// TIA Portal V17 export
// export: Created 2024-06-14T09:52:24.0418538Z, ExportSetting WithDefaults, DisplayName Totally Integrated Automation Portal, DisplayVersion V17, DisplayName TIA Portal Openness, DisplayVersion V17, DisplayName TIA Portal Version Control Interface, DisplayVersion V17, DisplayName Simotion SCOUT TIA, DisplayVersion 5.4.3.0, DisplayName SINAMICS Startdrive Advanced, DisplayVersion V17 SP1 Update 1, DisplayName SINAMICS Startdrive G110M, G120, G120C, G120D, G120P, G115D, DisplayVersion V17 SP1 Update 1, DisplayName SINAMICS Startdrive G130, G150, S120, S150, SINAMICS MV, S210, DisplayVersion V17 SP1 Update 1, DisplayName STEP 7 Professional, DisplayVersion V17, DisplayName STEP 7 Safety, DisplayVersion V17, DisplayName WinCC Professional, DisplayVersion V17
FUNCTION_BLOCK "TCP_STN4_STN2_FB"   // FB120, LAD
{ S7_Optimized_Access := 'TRUE' }
VERSION : 0.1
// stored: AutoNumber false, IsIECCheckEnabled false, IsRetainMemResEnabled false, MemoryReserve 100, SetENOAutomatically false, UDAEnableTagReadback false
   VAR_OUTPUT
      Modbus_Busy : Bool;
   END_VAR
   VAR_IN_OUT
      Mod_TCP_Setup : "Mod_TCP_Data";
      LPG_Fill_Data : "LPG_FILL_DATA";
   END_VAR
   VAR
      PStep_No : Struct
         MASTER_STEP_NO : "Master_Step_No";
      END_STRUCT;
      Write_Bit_Address : Int;
      TRIG : Array[1..100] of Bool;
      Mod_Master1_Req : Array[1..10] of Bool;
      Mod_Master2_REQ : Array[1..10] of Bool;
      Mod_Master3_REQ : Array[1..10] of Bool;
      Mod_Master4_REQ : Array[1..10] of Bool;
      Mod_Master5_REQ : Array[1..10] of Bool;
      Mod_Master6_REQ : Array[1..10] of Bool;
      Mas_Trig_Extn { S7_SetPoint := 'True'} : TOF_TIME;
      Tare_delay { S7_SetPoint := 'True'} : TON_TIME;
   END_VAR
   VAR_TEMP
      Modbus_request : Bool;
   END_VAR
   VAR_TEMP   // added for the SCL form of the ladder/FBD networks
      _w1 : Bool;
      _w2 : Bool;
      _w3 : Bool;
      _w4 : Bool;
      _w5 : Bool;
      _w6 : Bool;
   END_VAR
BEGIN

REGION Network 1: FILLING LINE-1 STATION-2
END_REGION

REGION Network 2: Write Master-1 Holding Register Request(Tare Weight Entry)
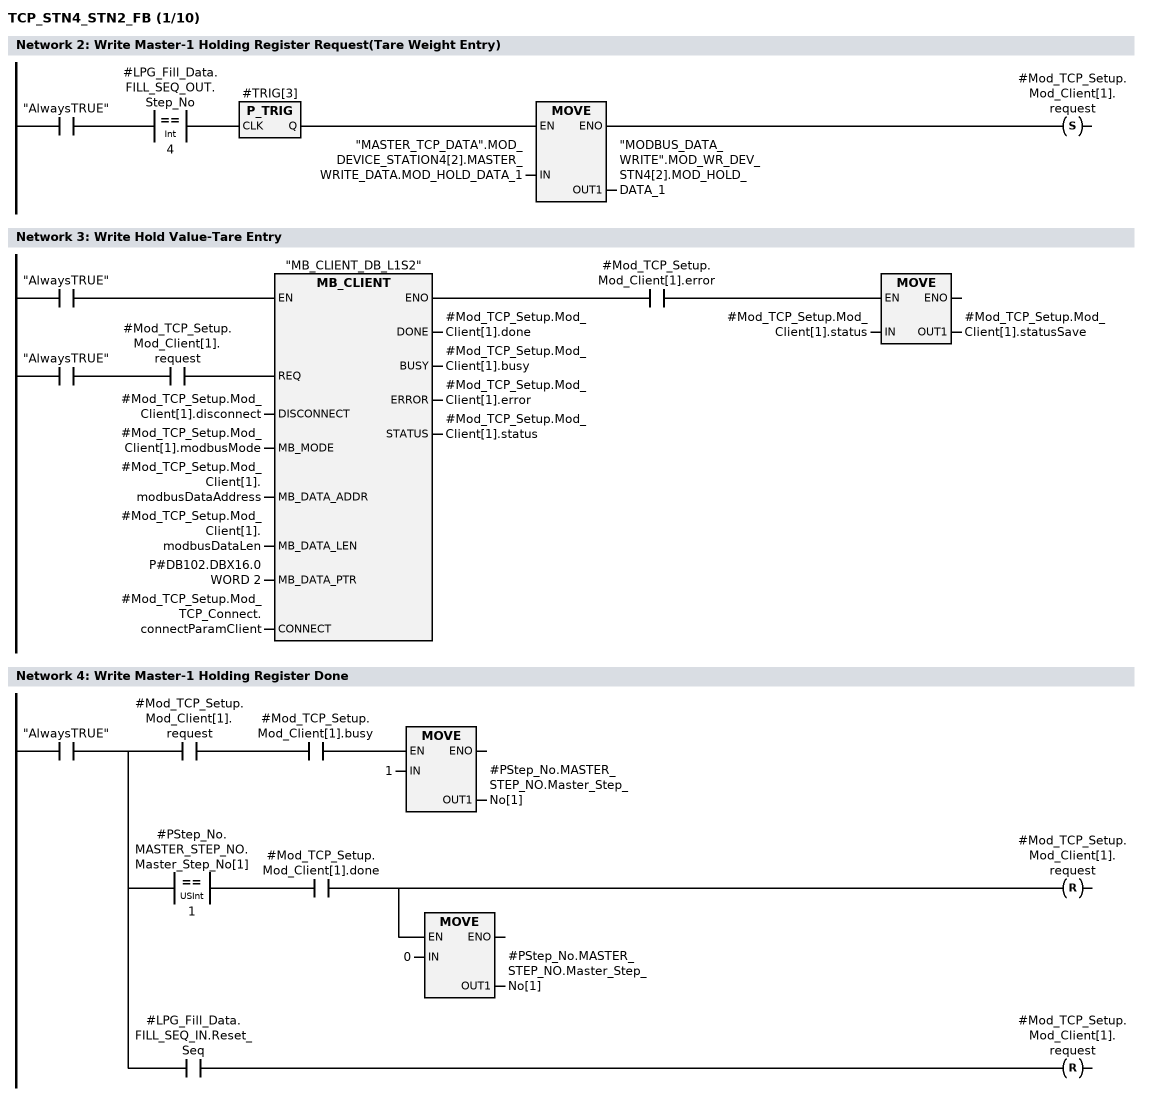
   RUNG wire#powerrail
      Contact( "AlwaysTRUE" )
      { S7_Templates := "SrcType := Int" } EQ_Contact(in1 := #LPG_Fill_Data.FILL_SEQ_OUT.Step_No, in2 := 4)
      P_Trig( #TRIG[3] )
      Move(in := "MASTER_TCP_DATA".MOD_DEVICE_STATION4[2].MASTER_WRITE_DATA.MOD_HOLD_DATA_1, out1 => "MODBUS_DATA_WRITE".MOD_WR_DEV_STN4[2].MOD_HOLD_DATA_1)
      S_Coil( #Mod_TCP_Setup.Mod_Client[1].request )
   END_RUNG
   // the same network as SCL:
   #_w1 := "AlwaysTRUE" AND (#LPG_Fill_Data.FILL_SEQ_OUT.Step_No = 4);
   #_w2 := #_w1 AND NOT #TRIG[3];   // rising edge
   #TRIG[3] := #_w1;
   IF #_w2 THEN
       "MODBUS_DATA_WRITE".MOD_WR_DEV_STN4[2].MOD_HOLD_DATA_1 := "MASTER_TCP_DATA".MOD_DEVICE_STATION4[2].MASTER_WRITE_DATA.MOD_HOLD_DATA_1;
       #Mod_TCP_Setup.Mod_Client[1].request := TRUE;
   END_IF;
END_REGION

REGION Network 3: Write Hold Value-Tare Entry
   RUNG wire#powerrail
      Contact( "AlwaysTRUE" )
      "MB_CLIENT_DB_L1S2".MB_CLIENT(REQ := wire#w1, DISCONNECT := #Mod_TCP_Setup.Mod_Client[1].disconnect, MB_MODE := #Mod_TCP_Setup.Mod_Client[1].modbusMode, MB_DATA_ADDR := #Mod_TCP_Setup.Mod_Client[1].modbusDataAddress, MB_DATA_LEN := #Mod_TCP_Setup.Mod_Client[1].modbusDataLen, MB_DATA_PTR := P#DB102.DBX16.0 WORD 2, CONNECT := #Mod_TCP_Setup.Mod_TCP_Connect.connectParamClient, DONE => #Mod_TCP_Setup.Mod_Client[1].done, BUSY => #Mod_TCP_Setup.Mod_Client[1].busy, ERROR => #Mod_TCP_Setup.Mod_Client[1].error, STATUS => #Mod_TCP_Setup.Mod_Client[1].status)
      Contact( #Mod_TCP_Setup.Mod_Client[1].error )
      Move(in := #Mod_TCP_Setup.Mod_Client[1].status, out1 => #Mod_TCP_Setup.Mod_Client[1].statusSave)
   END_RUNG
   RUNG wire#powerrail
      Contact( "AlwaysTRUE" )
      Contact( #Mod_TCP_Setup.Mod_Client[1].request )
   END_RUNG wire#w1
   // the same network as SCL:
   "MB_CLIENT_DB_L1S2"(EN := "AlwaysTRUE",   // MB_CLIENT
                       REQ := "AlwaysTRUE" AND #Mod_TCP_Setup.Mod_Client[1].request,
                       DISCONNECT := #Mod_TCP_Setup.Mod_Client[1].disconnect,
                       MB_MODE := #Mod_TCP_Setup.Mod_Client[1].modbusMode,
                       MB_DATA_ADDR := #Mod_TCP_Setup.Mod_Client[1].modbusDataAddress,
                       MB_DATA_LEN := #Mod_TCP_Setup.Mod_Client[1].modbusDataLen,
                       MB_DATA_PTR := P#DB102.DBX16.0 WORD 2,
                       CONNECT := #Mod_TCP_Setup.Mod_TCP_Connect.connectParamClient,
                       DONE => #Mod_TCP_Setup.Mod_Client[1].done,
                       BUSY => #Mod_TCP_Setup.Mod_Client[1].busy,
                       ERROR => #Mod_TCP_Setup.Mod_Client[1].error,
                       STATUS => #Mod_TCP_Setup.Mod_Client[1].status,
                       ENO => #_w1);
   IF #_w1 AND #Mod_TCP_Setup.Mod_Client[1].error THEN
       #Mod_TCP_Setup.Mod_Client[1].statusSave := #Mod_TCP_Setup.Mod_Client[1].status;
   END_IF;
END_REGION

REGION Network 4: Write Master-1 Holding Register Done
   RUNG wire#powerrail
      Contact( "AlwaysTRUE" )
      wire#w1
      Contact( #Mod_TCP_Setup.Mod_Client[1].request )
      Contact( #Mod_TCP_Setup.Mod_Client[1].busy )
      Move(in := 1, out1 => #PStep_No.MASTER_STEP_NO.Master_Step_No[1])
   END_RUNG
   RUNG wire#w1
      { S7_Templates := "SrcType := USInt" } EQ_Contact(in1 := #PStep_No.MASTER_STEP_NO.Master_Step_No[1], in2 := 1)
      Contact( #Mod_TCP_Setup.Mod_Client[1].done )
      wire#w2
      R_Coil( #Mod_TCP_Setup.Mod_Client[1].request )
   END_RUNG
   RUNG wire#w2
      Move(in := 0, out1 => #PStep_No.MASTER_STEP_NO.Master_Step_No[1])
   END_RUNG
   RUNG wire#w1
      Contact( #LPG_Fill_Data.FILL_SEQ_IN.Reset_Seq )
      R_Coil( #Mod_TCP_Setup.Mod_Client[1].request )
   END_RUNG
   // the same network as SCL:
   IF "AlwaysTRUE" AND #Mod_TCP_Setup.Mod_Client[1].request AND #Mod_TCP_Setup.Mod_Client[1].busy THEN
       #PStep_No.MASTER_STEP_NO.Master_Step_No[1] := 1;
   END_IF;
   #_w1 := "AlwaysTRUE" AND (#PStep_No.MASTER_STEP_NO.Master_Step_No[1] = 1) AND #Mod_TCP_Setup.Mod_Client[1].done;
   IF #_w1 THEN
       #Mod_TCP_Setup.Mod_Client[1].request := FALSE;
       #PStep_No.MASTER_STEP_NO.Master_Step_No[1] := 0;
   END_IF;
   IF "AlwaysTRUE" AND #LPG_Fill_Data.FILL_SEQ_IN.Reset_Seq THEN
       #Mod_TCP_Setup.Mod_Client[1].request := FALSE;
   END_IF;
END_REGION

REGION Network 5: Modbus Master2 Read Request(Filled Data)
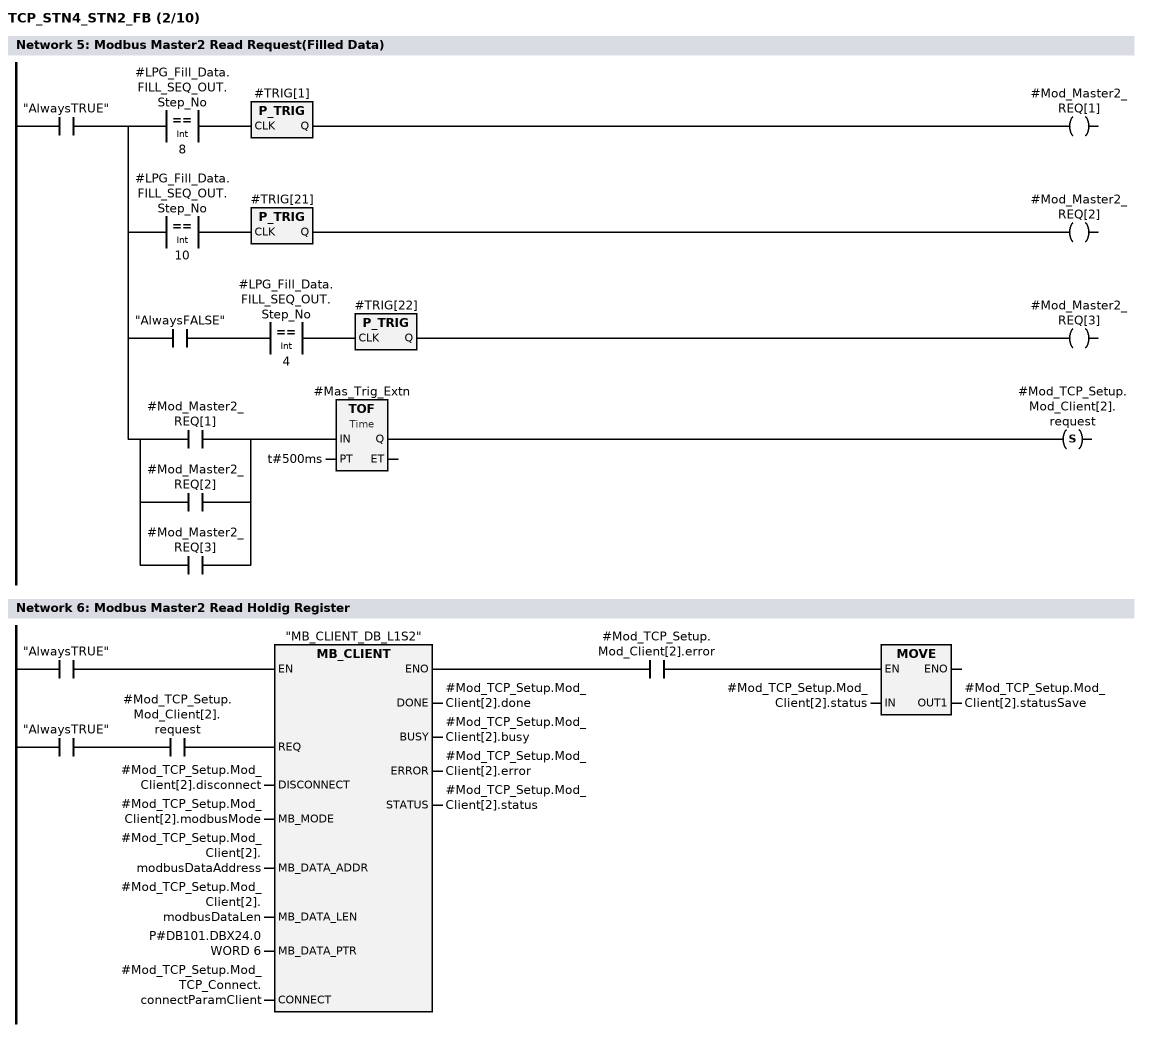
   RUNG wire#powerrail
      Contact( "AlwaysTRUE" )
      wire#w1
      { S7_Templates := "SrcType := Int" } EQ_Contact(in1 := #LPG_Fill_Data.FILL_SEQ_OUT.Step_No, in2 := 8)
      P_Trig( #TRIG[1] )
      Coil( #Mod_Master2_REQ[1] )
   END_RUNG
   RUNG wire#w1
      { S7_Templates := "SrcType := Int" } EQ_Contact(in1 := #LPG_Fill_Data.FILL_SEQ_OUT.Step_No, in2 := 10)
      P_Trig( #TRIG[21] )
      Coil( #Mod_Master2_REQ[2] )
   END_RUNG
   RUNG wire#w1
      Contact( "AlwaysFALSE" )
      { S7_Templates := "SrcType := Int" } EQ_Contact(in1 := #LPG_Fill_Data.FILL_SEQ_OUT.Step_No, in2 := 4)
      P_Trig( #TRIG[22] )
      Coil( #Mod_Master2_REQ[3] )
   END_RUNG
   RUNG wire#w1
      Contact( #Mod_Master2_REQ[1] )
      wire#w2
      { S7_Templates := "time_type := Time" } #Mas_Trig_Extn.TOF(pt := t#500ms, et =>)
      S_Coil( #Mod_TCP_Setup.Mod_Client[2].request )
   END_RUNG
   RUNG wire#w1
      Contact( #Mod_Master2_REQ[2] )
   END_RUNG wire#w2
   RUNG wire#w1
      Contact( #Mod_Master2_REQ[3] )
   END_RUNG wire#w2
   // the same network as SCL:
   #_w1 := "AlwaysTRUE" AND (#LPG_Fill_Data.FILL_SEQ_OUT.Step_No = 8);
   #_w2 := #_w1 AND NOT #TRIG[1];   // rising edge
   #TRIG[1] := #_w1;
   #Mod_Master2_REQ[1] := #_w2;
   #_w3 := "AlwaysTRUE" AND (#LPG_Fill_Data.FILL_SEQ_OUT.Step_No = 10);
   #_w4 := #_w3 AND NOT #TRIG[21];   // rising edge
   #TRIG[21] := #_w3;
   #Mod_Master2_REQ[2] := #_w4;
   #_w5 := "AlwaysTRUE" AND "AlwaysFALSE" AND (#LPG_Fill_Data.FILL_SEQ_OUT.Step_No = 4);
   #_w6 := #_w5 AND NOT #TRIG[22];   // rising edge
   #TRIG[22] := #_w5;
   #Mod_Master2_REQ[3] := #_w6;
   #Mas_Trig_Extn(IN := "AlwaysTRUE" AND (#Mod_Master2_REQ[1] OR #Mod_Master2_REQ[2] OR #Mod_Master2_REQ[3]),   // TOF
                  PT := t#500ms);
   IF #Mas_Trig_Extn.Q THEN #Mod_TCP_Setup.Mod_Client[2].request := TRUE; END_IF;
END_REGION

REGION Network 6: Modbus Master2 Read Holdig Register
   RUNG wire#powerrail
      Contact( "AlwaysTRUE" )
      "MB_CLIENT_DB_L1S2".MB_CLIENT(REQ := wire#w1, DISCONNECT := #Mod_TCP_Setup.Mod_Client[2].disconnect, MB_MODE := #Mod_TCP_Setup.Mod_Client[2].modbusMode, MB_DATA_ADDR := #Mod_TCP_Setup.Mod_Client[2].modbusDataAddress, MB_DATA_LEN := #Mod_TCP_Setup.Mod_Client[2].modbusDataLen, MB_DATA_PTR := P#DB101.DBX24.0 WORD 6, CONNECT := #Mod_TCP_Setup.Mod_TCP_Connect.connectParamClient, DONE => #Mod_TCP_Setup.Mod_Client[2].done, BUSY => #Mod_TCP_Setup.Mod_Client[2].busy, ERROR => #Mod_TCP_Setup.Mod_Client[2].error, STATUS => #Mod_TCP_Setup.Mod_Client[2].status)
      Contact( #Mod_TCP_Setup.Mod_Client[2].error )
      Move(in := #Mod_TCP_Setup.Mod_Client[2].status, out1 => #Mod_TCP_Setup.Mod_Client[2].statusSave)
   END_RUNG
   RUNG wire#powerrail
      Contact( "AlwaysTRUE" )
      Contact( #Mod_TCP_Setup.Mod_Client[2].request )
   END_RUNG wire#w1
   // the same network as SCL:
   "MB_CLIENT_DB_L1S2"(EN := "AlwaysTRUE",   // MB_CLIENT
                       REQ := "AlwaysTRUE" AND #Mod_TCP_Setup.Mod_Client[2].request,
                       DISCONNECT := #Mod_TCP_Setup.Mod_Client[2].disconnect,
                       MB_MODE := #Mod_TCP_Setup.Mod_Client[2].modbusMode,
                       MB_DATA_ADDR := #Mod_TCP_Setup.Mod_Client[2].modbusDataAddress,
                       MB_DATA_LEN := #Mod_TCP_Setup.Mod_Client[2].modbusDataLen,
                       MB_DATA_PTR := P#DB101.DBX24.0 WORD 6,
                       CONNECT := #Mod_TCP_Setup.Mod_TCP_Connect.connectParamClient,
                       DONE => #Mod_TCP_Setup.Mod_Client[2].done,
                       BUSY => #Mod_TCP_Setup.Mod_Client[2].busy,
                       ERROR => #Mod_TCP_Setup.Mod_Client[2].error,
                       STATUS => #Mod_TCP_Setup.Mod_Client[2].status,
                       ENO => #_w1);
   IF #_w1 AND #Mod_TCP_Setup.Mod_Client[2].error THEN
       #Mod_TCP_Setup.Mod_Client[2].statusSave := #Mod_TCP_Setup.Mod_Client[2].status;
   END_IF;
END_REGION

REGION Network 7: Read Master-2 Holding Register Value
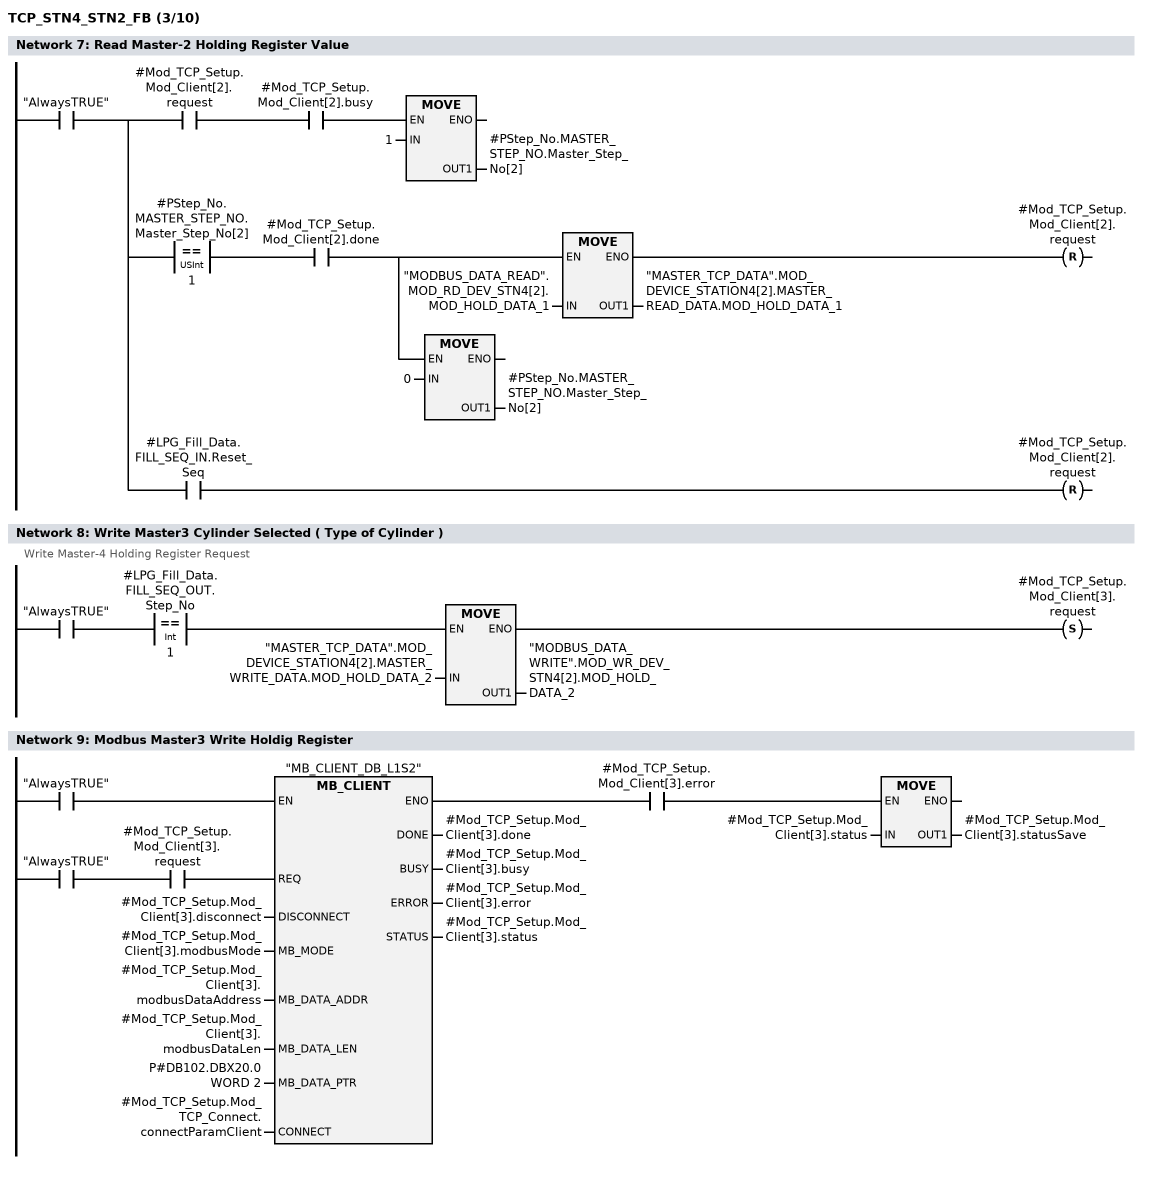
   RUNG wire#powerrail
      Contact( "AlwaysTRUE" )
      wire#w1
      Contact( #Mod_TCP_Setup.Mod_Client[2].request )
      Contact( #Mod_TCP_Setup.Mod_Client[2].busy )
      Move(in := 1, out1 => #PStep_No.MASTER_STEP_NO.Master_Step_No[2])
   END_RUNG
   RUNG wire#w1
      { S7_Templates := "SrcType := USInt" } EQ_Contact(in1 := #PStep_No.MASTER_STEP_NO.Master_Step_No[2], in2 := 1)
      Contact( #Mod_TCP_Setup.Mod_Client[2].done )
      wire#w2
      Move(in := "MODBUS_DATA_READ".MOD_RD_DEV_STN4[2].MOD_HOLD_DATA_1, out1 => "MASTER_TCP_DATA".MOD_DEVICE_STATION4[2].MASTER_READ_DATA.MOD_HOLD_DATA_1)
      R_Coil( #Mod_TCP_Setup.Mod_Client[2].request )
   END_RUNG
   RUNG wire#w2
      Move(in := 0, out1 => #PStep_No.MASTER_STEP_NO.Master_Step_No[2])
   END_RUNG
   RUNG wire#w1
      Contact( #LPG_Fill_Data.FILL_SEQ_IN.Reset_Seq )
      R_Coil( #Mod_TCP_Setup.Mod_Client[2].request )
   END_RUNG
   // the same network as SCL:
   IF "AlwaysTRUE" AND #Mod_TCP_Setup.Mod_Client[2].request AND #Mod_TCP_Setup.Mod_Client[2].busy THEN
       #PStep_No.MASTER_STEP_NO.Master_Step_No[2] := 1;
   END_IF;
   IF "AlwaysTRUE" AND (#PStep_No.MASTER_STEP_NO.Master_Step_No[2] = 1) AND #Mod_TCP_Setup.Mod_Client[2].done THEN
       "MASTER_TCP_DATA".MOD_DEVICE_STATION4[2].MASTER_READ_DATA.MOD_HOLD_DATA_1 := "MODBUS_DATA_READ".MOD_RD_DEV_STN4[2].MOD_HOLD_DATA_1;
   END_IF;
   #_w1 := "AlwaysTRUE" AND (#PStep_No.MASTER_STEP_NO.Master_Step_No[2] = 1) AND #Mod_TCP_Setup.Mod_Client[2].done;
   IF #_w1 THEN
       #Mod_TCP_Setup.Mod_Client[2].request := FALSE;
       #PStep_No.MASTER_STEP_NO.Master_Step_No[2] := 0;
   END_IF;
   IF "AlwaysTRUE" AND #LPG_Fill_Data.FILL_SEQ_IN.Reset_Seq THEN
       #Mod_TCP_Setup.Mod_Client[2].request := FALSE;
   END_IF;
END_REGION

REGION Network 8: Write Master3 Cylinder Selected ( Type of Cylinder )
   // Write Master-4 Holding Register Request
   RUNG wire#powerrail
      Contact( "AlwaysTRUE" )
      { S7_Templates := "SrcType := Int" } EQ_Contact(in1 := #LPG_Fill_Data.FILL_SEQ_OUT.Step_No, in2 := 1)
      Move(in := "MASTER_TCP_DATA".MOD_DEVICE_STATION4[2].MASTER_WRITE_DATA.MOD_HOLD_DATA_2, out1 => "MODBUS_DATA_WRITE".MOD_WR_DEV_STN4[2].MOD_HOLD_DATA_2)
      S_Coil( #Mod_TCP_Setup.Mod_Client[3].request )
   END_RUNG
   // the same network as SCL:
   IF "AlwaysTRUE" AND (#LPG_Fill_Data.FILL_SEQ_OUT.Step_No = 1) THEN
       "MODBUS_DATA_WRITE".MOD_WR_DEV_STN4[2].MOD_HOLD_DATA_2 := "MASTER_TCP_DATA".MOD_DEVICE_STATION4[2].MASTER_WRITE_DATA.MOD_HOLD_DATA_2;
       #Mod_TCP_Setup.Mod_Client[3].request := TRUE;
   END_IF;
END_REGION

REGION Network 9: Modbus Master3 Write Holdig Register
   RUNG wire#powerrail
      Contact( "AlwaysTRUE" )
      "MB_CLIENT_DB_L1S2".MB_CLIENT(REQ := wire#w1, DISCONNECT := #Mod_TCP_Setup.Mod_Client[3].disconnect, MB_MODE := #Mod_TCP_Setup.Mod_Client[3].modbusMode, MB_DATA_ADDR := #Mod_TCP_Setup.Mod_Client[3].modbusDataAddress, MB_DATA_LEN := #Mod_TCP_Setup.Mod_Client[3].modbusDataLen, MB_DATA_PTR := P#DB102.DBX20.0 WORD 2, CONNECT := #Mod_TCP_Setup.Mod_TCP_Connect.connectParamClient, DONE => #Mod_TCP_Setup.Mod_Client[3].done, BUSY => #Mod_TCP_Setup.Mod_Client[3].busy, ERROR => #Mod_TCP_Setup.Mod_Client[3].error, STATUS => #Mod_TCP_Setup.Mod_Client[3].status)
      Contact( #Mod_TCP_Setup.Mod_Client[3].error )
      Move(in := #Mod_TCP_Setup.Mod_Client[3].status, out1 => #Mod_TCP_Setup.Mod_Client[3].statusSave)
   END_RUNG
   RUNG wire#powerrail
      Contact( "AlwaysTRUE" )
      Contact( #Mod_TCP_Setup.Mod_Client[3].request )
   END_RUNG wire#w1
   // the same network as SCL:
   "MB_CLIENT_DB_L1S2"(EN := "AlwaysTRUE",   // MB_CLIENT
                       REQ := "AlwaysTRUE" AND #Mod_TCP_Setup.Mod_Client[3].request,
                       DISCONNECT := #Mod_TCP_Setup.Mod_Client[3].disconnect,
                       MB_MODE := #Mod_TCP_Setup.Mod_Client[3].modbusMode,
                       MB_DATA_ADDR := #Mod_TCP_Setup.Mod_Client[3].modbusDataAddress,
                       MB_DATA_LEN := #Mod_TCP_Setup.Mod_Client[3].modbusDataLen,
                       MB_DATA_PTR := P#DB102.DBX20.0 WORD 2,
                       CONNECT := #Mod_TCP_Setup.Mod_TCP_Connect.connectParamClient,
                       DONE => #Mod_TCP_Setup.Mod_Client[3].done,
                       BUSY => #Mod_TCP_Setup.Mod_Client[3].busy,
                       ERROR => #Mod_TCP_Setup.Mod_Client[3].error,
                       STATUS => #Mod_TCP_Setup.Mod_Client[3].status,
                       ENO => #_w1);
   IF #_w1 AND #Mod_TCP_Setup.Mod_Client[3].error THEN
       #Mod_TCP_Setup.Mod_Client[3].statusSave := #Mod_TCP_Setup.Mod_Client[3].status;
   END_IF;
END_REGION

REGION Network 10: Write Master-3 Holding Register Done
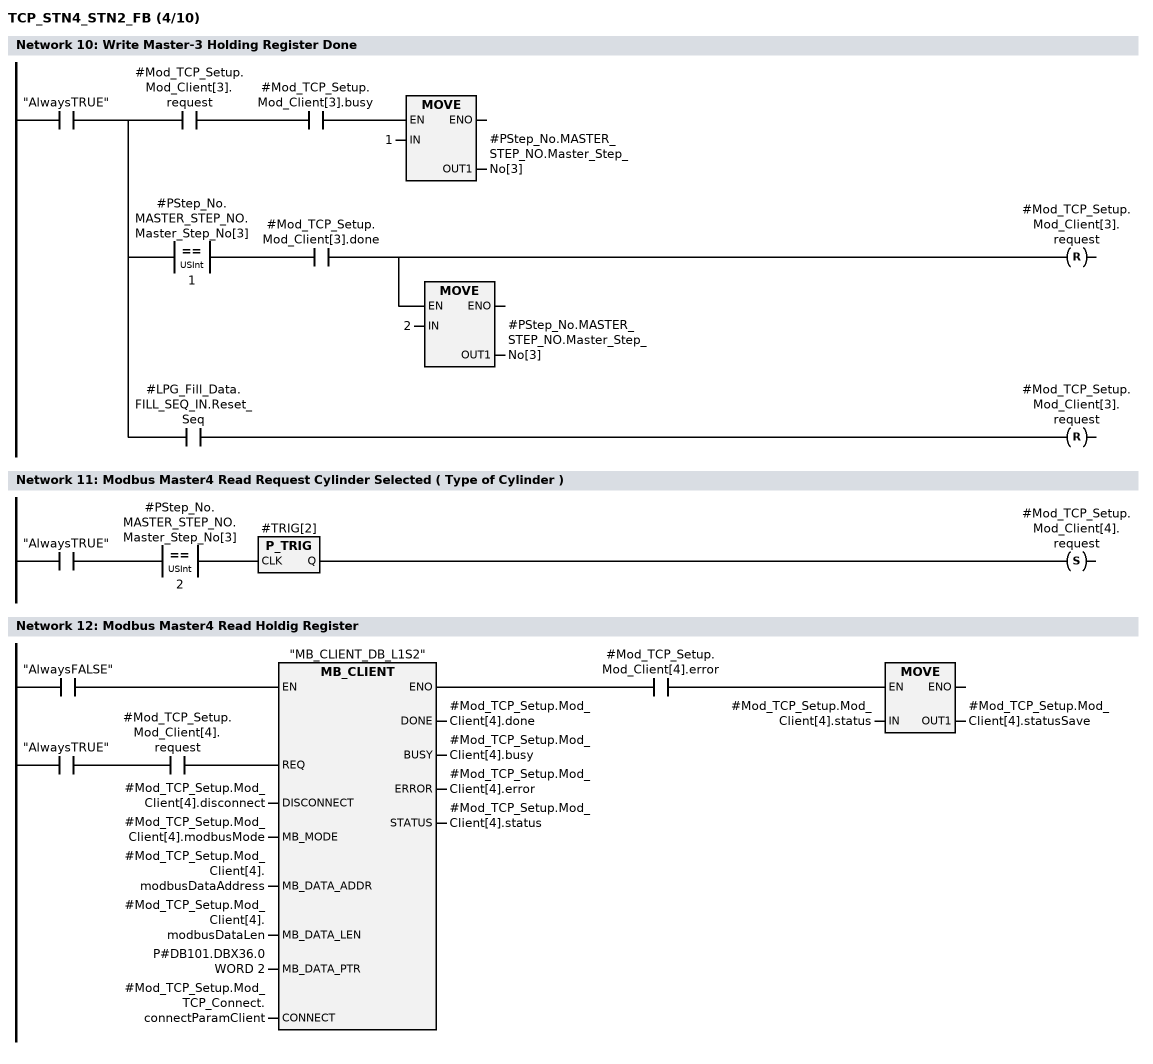
   RUNG wire#powerrail
      Contact( "AlwaysTRUE" )
      wire#w1
      Contact( #Mod_TCP_Setup.Mod_Client[3].request )
      Contact( #Mod_TCP_Setup.Mod_Client[3].busy )
      Move(in := 1, out1 => #PStep_No.MASTER_STEP_NO.Master_Step_No[3])
   END_RUNG
   RUNG wire#w1
      { S7_Templates := "SrcType := USInt" } EQ_Contact(in1 := #PStep_No.MASTER_STEP_NO.Master_Step_No[3], in2 := 1)
      Contact( #Mod_TCP_Setup.Mod_Client[3].done )
      wire#w2
      R_Coil( #Mod_TCP_Setup.Mod_Client[3].request )
   END_RUNG
   RUNG wire#w2
      Move(in := 2, out1 => #PStep_No.MASTER_STEP_NO.Master_Step_No[3])
   END_RUNG
   RUNG wire#w1
      Contact( #LPG_Fill_Data.FILL_SEQ_IN.Reset_Seq )
      R_Coil( #Mod_TCP_Setup.Mod_Client[3].request )
   END_RUNG
   // the same network as SCL:
   IF "AlwaysTRUE" AND #Mod_TCP_Setup.Mod_Client[3].request AND #Mod_TCP_Setup.Mod_Client[3].busy THEN
       #PStep_No.MASTER_STEP_NO.Master_Step_No[3] := 1;
   END_IF;
   #_w1 := "AlwaysTRUE" AND (#PStep_No.MASTER_STEP_NO.Master_Step_No[3] = 1) AND #Mod_TCP_Setup.Mod_Client[3].done;
   IF #_w1 THEN
       #Mod_TCP_Setup.Mod_Client[3].request := FALSE;
       #PStep_No.MASTER_STEP_NO.Master_Step_No[3] := 2;
   END_IF;
   IF "AlwaysTRUE" AND #LPG_Fill_Data.FILL_SEQ_IN.Reset_Seq THEN
       #Mod_TCP_Setup.Mod_Client[3].request := FALSE;
   END_IF;
END_REGION

REGION Network 11: Modbus Master4 Read Request Cylinder Selected ( Type of Cylinder )
   RUNG wire#powerrail
      Contact( "AlwaysTRUE" )
      { S7_Templates := "SrcType := USInt" } EQ_Contact(in1 := #PStep_No.MASTER_STEP_NO.Master_Step_No[3], in2 := 2)
      P_Trig( #TRIG[2] )
      S_Coil( #Mod_TCP_Setup.Mod_Client[4].request )
   END_RUNG
   // the same network as SCL:
   #_w1 := "AlwaysTRUE" AND (#PStep_No.MASTER_STEP_NO.Master_Step_No[3] = 2);
   #_w2 := #_w1 AND NOT #TRIG[2];   // rising edge
   #TRIG[2] := #_w1;
   IF #_w2 THEN #Mod_TCP_Setup.Mod_Client[4].request := TRUE; END_IF;
END_REGION

REGION Network 12: Modbus Master4 Read Holdig Register
   RUNG wire#powerrail
      Contact( "AlwaysFALSE" )
      "MB_CLIENT_DB_L1S2".MB_CLIENT(REQ := wire#w1, DISCONNECT := #Mod_TCP_Setup.Mod_Client[4].disconnect, MB_MODE := #Mod_TCP_Setup.Mod_Client[4].modbusMode, MB_DATA_ADDR := #Mod_TCP_Setup.Mod_Client[4].modbusDataAddress, MB_DATA_LEN := #Mod_TCP_Setup.Mod_Client[4].modbusDataLen, MB_DATA_PTR := P#DB101.DBX36.0 WORD 2, CONNECT := #Mod_TCP_Setup.Mod_TCP_Connect.connectParamClient, DONE => #Mod_TCP_Setup.Mod_Client[4].done, BUSY => #Mod_TCP_Setup.Mod_Client[4].busy, ERROR => #Mod_TCP_Setup.Mod_Client[4].error, STATUS => #Mod_TCP_Setup.Mod_Client[4].status)
      Contact( #Mod_TCP_Setup.Mod_Client[4].error )
      Move(in := #Mod_TCP_Setup.Mod_Client[4].status, out1 => #Mod_TCP_Setup.Mod_Client[4].statusSave)
   END_RUNG
   RUNG wire#powerrail
      Contact( "AlwaysTRUE" )
      Contact( #Mod_TCP_Setup.Mod_Client[4].request )
   END_RUNG wire#w1
   // the same network as SCL:
   "MB_CLIENT_DB_L1S2"(EN := "AlwaysFALSE",   // MB_CLIENT
                       REQ := "AlwaysTRUE" AND #Mod_TCP_Setup.Mod_Client[4].request,
                       DISCONNECT := #Mod_TCP_Setup.Mod_Client[4].disconnect,
                       MB_MODE := #Mod_TCP_Setup.Mod_Client[4].modbusMode,
                       MB_DATA_ADDR := #Mod_TCP_Setup.Mod_Client[4].modbusDataAddress,
                       MB_DATA_LEN := #Mod_TCP_Setup.Mod_Client[4].modbusDataLen,
                       MB_DATA_PTR := P#DB101.DBX36.0 WORD 2,
                       CONNECT := #Mod_TCP_Setup.Mod_TCP_Connect.connectParamClient,
                       DONE => #Mod_TCP_Setup.Mod_Client[4].done,
                       BUSY => #Mod_TCP_Setup.Mod_Client[4].busy,
                       ERROR => #Mod_TCP_Setup.Mod_Client[4].error,
                       STATUS => #Mod_TCP_Setup.Mod_Client[4].status,
                       ENO => #_w1);
   IF #_w1 AND #Mod_TCP_Setup.Mod_Client[4].error THEN
       #Mod_TCP_Setup.Mod_Client[4].statusSave := #Mod_TCP_Setup.Mod_Client[4].status;
   END_IF;
END_REGION

REGION Network 13: Read Master-4 Holding Register Value
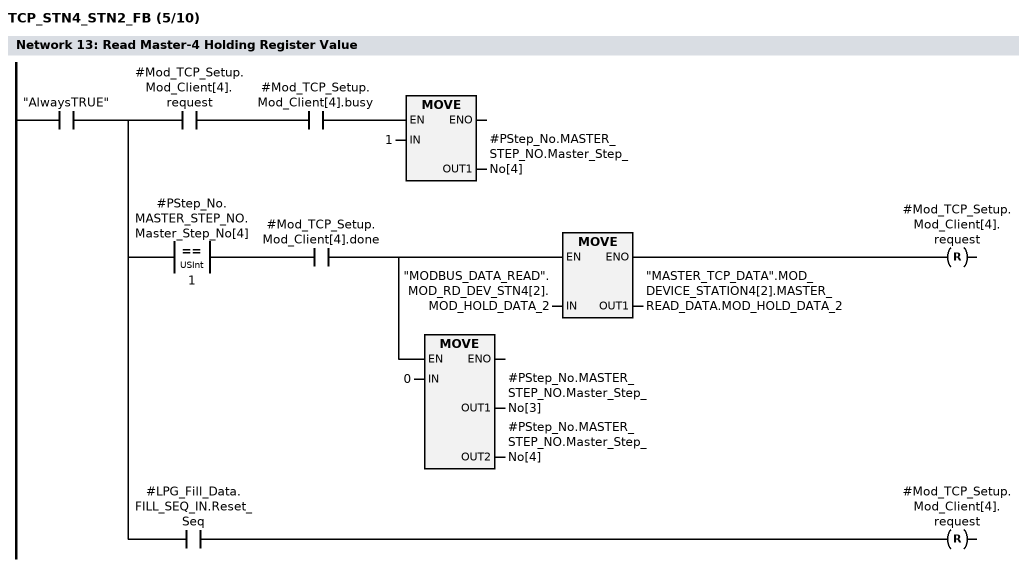
   RUNG wire#powerrail
      Contact( "AlwaysTRUE" )
      wire#w1
      Contact( #Mod_TCP_Setup.Mod_Client[4].request )
      Contact( #Mod_TCP_Setup.Mod_Client[4].busy )
      Move(in := 1, out1 => #PStep_No.MASTER_STEP_NO.Master_Step_No[4])
   END_RUNG
   RUNG wire#w1
      { S7_Templates := "SrcType := USInt" } EQ_Contact(in1 := #PStep_No.MASTER_STEP_NO.Master_Step_No[4], in2 := 1)
      Contact( #Mod_TCP_Setup.Mod_Client[4].done )
      wire#w2
      Move(in := "MODBUS_DATA_READ".MOD_RD_DEV_STN4[2].MOD_HOLD_DATA_2, out1 => "MASTER_TCP_DATA".MOD_DEVICE_STATION4[2].MASTER_READ_DATA.MOD_HOLD_DATA_2)
      R_Coil( #Mod_TCP_Setup.Mod_Client[4].request )
   END_RUNG
   RUNG wire#w2
      Move(in := 0, out1 => #PStep_No.MASTER_STEP_NO.Master_Step_No[3], out2 => #PStep_No.MASTER_STEP_NO.Master_Step_No[4])
   END_RUNG
   RUNG wire#w1
      Contact( #LPG_Fill_Data.FILL_SEQ_IN.Reset_Seq )
      R_Coil( #Mod_TCP_Setup.Mod_Client[4].request )
   END_RUNG
   // the same network as SCL:
   IF "AlwaysTRUE" AND #Mod_TCP_Setup.Mod_Client[4].request AND #Mod_TCP_Setup.Mod_Client[4].busy THEN
       #PStep_No.MASTER_STEP_NO.Master_Step_No[4] := 1;
   END_IF;
   IF "AlwaysTRUE" AND (#PStep_No.MASTER_STEP_NO.Master_Step_No[4] = 1) AND #Mod_TCP_Setup.Mod_Client[4].done THEN
       "MASTER_TCP_DATA".MOD_DEVICE_STATION4[2].MASTER_READ_DATA.MOD_HOLD_DATA_2 := "MODBUS_DATA_READ".MOD_RD_DEV_STN4[2].MOD_HOLD_DATA_2;
   END_IF;
   #_w1 := "AlwaysTRUE" AND (#PStep_No.MASTER_STEP_NO.Master_Step_No[4] = 1) AND #Mod_TCP_Setup.Mod_Client[4].done;
   IF #_w1 THEN
       #Mod_TCP_Setup.Mod_Client[4].request := FALSE;
       #PStep_No.MASTER_STEP_NO.Master_Step_No[3] := 0;
       #PStep_No.MASTER_STEP_NO.Master_Step_No[4] := 0;
   END_IF;
   IF "AlwaysTRUE" AND #LPG_Fill_Data.FILL_SEQ_IN.Reset_Seq THEN
       #Mod_TCP_Setup.Mod_Client[4].request := FALSE;
   END_IF;
END_REGION

REGION Network 14: Modbus Master5 Read Request(Coil Status)
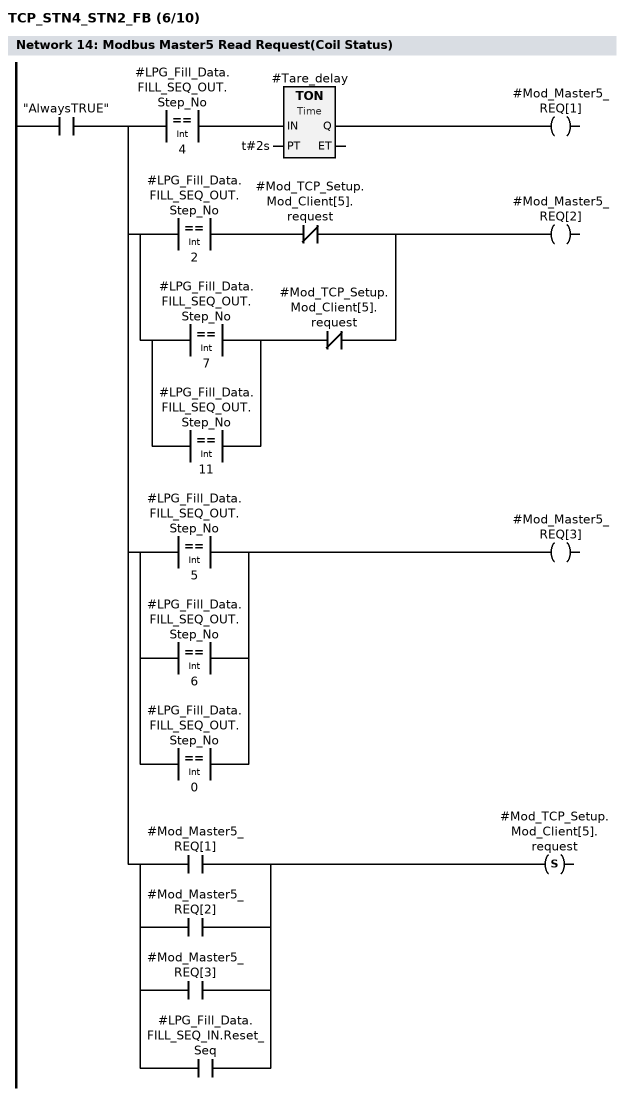
   RUNG wire#powerrail
      Contact( "AlwaysTRUE" )
      wire#w1
      { S7_Templates := "SrcType := Int" } EQ_Contact(in1 := #LPG_Fill_Data.FILL_SEQ_OUT.Step_No, in2 := 4)
      { S7_Templates := "time_type := Time" } #Tare_delay.TON(pt := t#2s, et =>)
      Coil( #Mod_Master5_REQ[1] )
   END_RUNG
   RUNG wire#w1
      { S7_Templates := "SrcType := Int" } EQ_Contact(in1 := #LPG_Fill_Data.FILL_SEQ_OUT.Step_No, in2 := 2)
      I_Contact( #Mod_TCP_Setup.Mod_Client[5].request )
      wire#w2
      Coil( #Mod_Master5_REQ[2] )
   END_RUNG
   RUNG wire#w1
      { S7_Templates := "SrcType := Int" } EQ_Contact(in1 := #LPG_Fill_Data.FILL_SEQ_OUT.Step_No, in2 := 7)
      wire#w3
      I_Contact( #Mod_TCP_Setup.Mod_Client[5].request )
   END_RUNG wire#w2
   RUNG wire#w1
      { S7_Templates := "SrcType := Int" } EQ_Contact(in1 := #LPG_Fill_Data.FILL_SEQ_OUT.Step_No, in2 := 11)
   END_RUNG wire#w3
   RUNG wire#w1
      { S7_Templates := "SrcType := Int" } EQ_Contact(in1 := #LPG_Fill_Data.FILL_SEQ_OUT.Step_No, in2 := 5)
      wire#w4
      Coil( #Mod_Master5_REQ[3] )
   END_RUNG
   RUNG wire#w1
      { S7_Templates := "SrcType := Int" } EQ_Contact(in1 := #LPG_Fill_Data.FILL_SEQ_OUT.Step_No, in2 := 6)
   END_RUNG wire#w4
   RUNG wire#w1
      { S7_Templates := "SrcType := Int" } EQ_Contact(in1 := #LPG_Fill_Data.FILL_SEQ_OUT.Step_No, in2 := 0)
   END_RUNG wire#w4
   RUNG wire#w1
      Contact( #Mod_Master5_REQ[1] )
      wire#w5
      S_Coil( #Mod_TCP_Setup.Mod_Client[5].request )
   END_RUNG
   RUNG wire#w1
      Contact( #Mod_Master5_REQ[2] )
   END_RUNG wire#w5
   RUNG wire#w1
      Contact( #Mod_Master5_REQ[3] )
   END_RUNG wire#w5
   RUNG wire#w1
      Contact( #LPG_Fill_Data.FILL_SEQ_IN.Reset_Seq )
   END_RUNG wire#w5
   // the same network as SCL:
   #Tare_delay(IN := "AlwaysTRUE" AND (#LPG_Fill_Data.FILL_SEQ_OUT.Step_No = 4), PT := t#2s);   // TON
   #Mod_Master5_REQ[1] := #Tare_delay.Q;
   #Mod_Master5_REQ[2] := "AlwaysTRUE" AND (((#LPG_Fill_Data.FILL_SEQ_OUT.Step_No = 2) AND NOT #Mod_TCP_Setup.Mod_Client[5].request) OR (((#LPG_Fill_Data.FILL_SEQ_OUT.Step_No = 7) OR (#LPG_Fill_Data.FILL_SEQ_OUT.Step_No = 11)) AND NOT #Mod_TCP_Setup.Mod_Client[5].request));
   #Mod_Master5_REQ[3] := "AlwaysTRUE" AND ((#LPG_Fill_Data.FILL_SEQ_OUT.Step_No = 5) OR (#LPG_Fill_Data.FILL_SEQ_OUT.Step_No = 6) OR (#LPG_Fill_Data.FILL_SEQ_OUT.Step_No = 0));
   IF "AlwaysTRUE" AND (#Mod_Master5_REQ[1] OR #Mod_Master5_REQ[2] OR #Mod_Master5_REQ[3] OR #LPG_Fill_Data.FILL_SEQ_IN.Reset_Seq) THEN
       #Mod_TCP_Setup.Mod_Client[5].request := TRUE;
   END_IF;
END_REGION

REGION Network 15: Modbus Master5 Read Coil Status
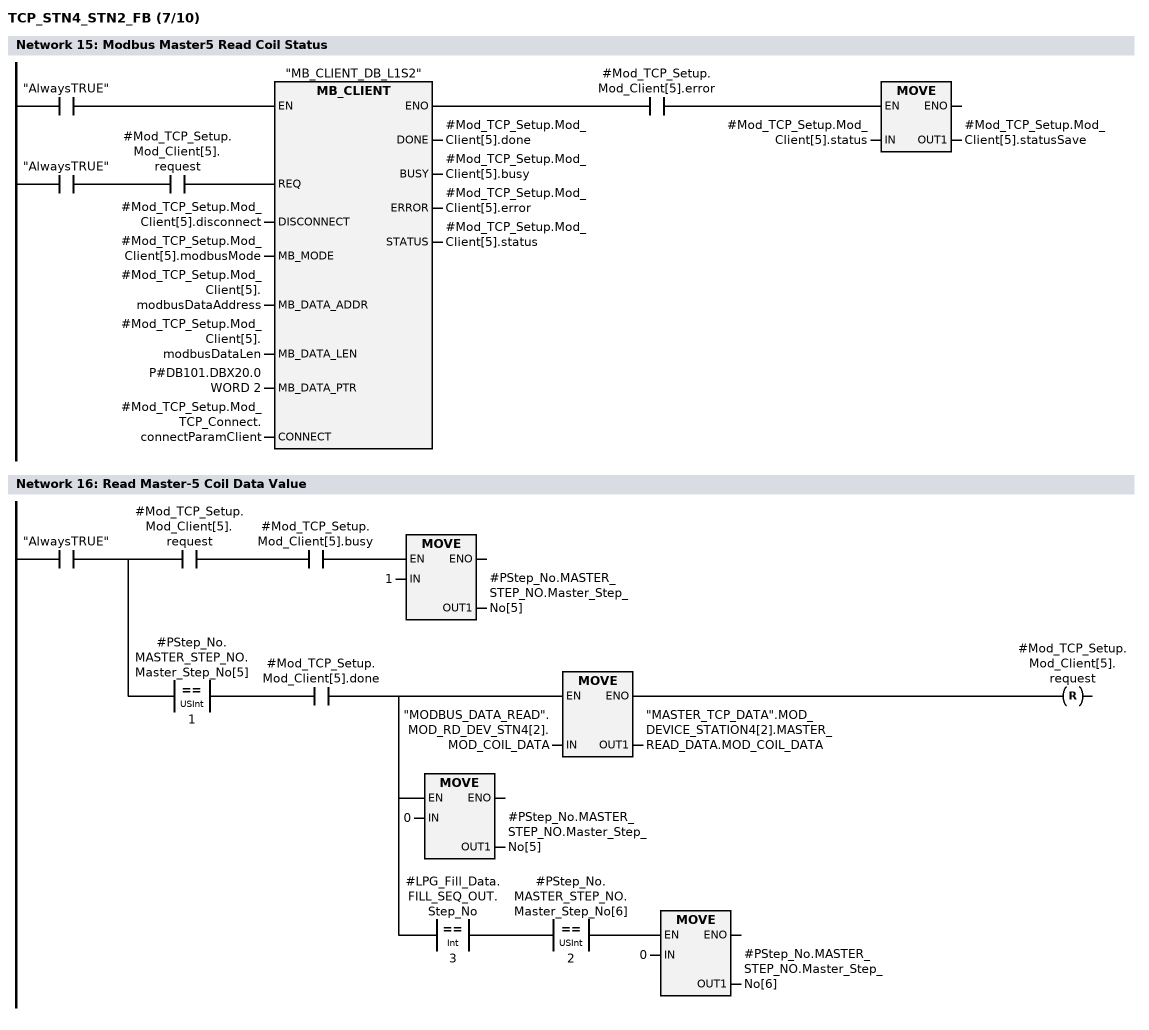
   RUNG wire#powerrail
      Contact( "AlwaysTRUE" )
      "MB_CLIENT_DB_L1S2".MB_CLIENT(REQ := wire#w1, DISCONNECT := #Mod_TCP_Setup.Mod_Client[5].disconnect, MB_MODE := #Mod_TCP_Setup.Mod_Client[5].modbusMode, MB_DATA_ADDR := #Mod_TCP_Setup.Mod_Client[5].modbusDataAddress, MB_DATA_LEN := #Mod_TCP_Setup.Mod_Client[5].modbusDataLen, MB_DATA_PTR := P#DB101.DBX20.0 WORD 2, CONNECT := #Mod_TCP_Setup.Mod_TCP_Connect.connectParamClient, DONE => #Mod_TCP_Setup.Mod_Client[5].done, BUSY => #Mod_TCP_Setup.Mod_Client[5].busy, ERROR => #Mod_TCP_Setup.Mod_Client[5].error, STATUS => #Mod_TCP_Setup.Mod_Client[5].status)
      Contact( #Mod_TCP_Setup.Mod_Client[5].error )
      Move(in := #Mod_TCP_Setup.Mod_Client[5].status, out1 => #Mod_TCP_Setup.Mod_Client[5].statusSave)
   END_RUNG
   RUNG wire#powerrail
      Contact( "AlwaysTRUE" )
      Contact( #Mod_TCP_Setup.Mod_Client[5].request )
   END_RUNG wire#w1
   // the same network as SCL:
   "MB_CLIENT_DB_L1S2"(EN := "AlwaysTRUE",   // MB_CLIENT
                       REQ := "AlwaysTRUE" AND #Mod_TCP_Setup.Mod_Client[5].request,
                       DISCONNECT := #Mod_TCP_Setup.Mod_Client[5].disconnect,
                       MB_MODE := #Mod_TCP_Setup.Mod_Client[5].modbusMode,
                       MB_DATA_ADDR := #Mod_TCP_Setup.Mod_Client[5].modbusDataAddress,
                       MB_DATA_LEN := #Mod_TCP_Setup.Mod_Client[5].modbusDataLen,
                       MB_DATA_PTR := P#DB101.DBX20.0 WORD 2,
                       CONNECT := #Mod_TCP_Setup.Mod_TCP_Connect.connectParamClient,
                       DONE => #Mod_TCP_Setup.Mod_Client[5].done,
                       BUSY => #Mod_TCP_Setup.Mod_Client[5].busy,
                       ERROR => #Mod_TCP_Setup.Mod_Client[5].error,
                       STATUS => #Mod_TCP_Setup.Mod_Client[5].status,
                       ENO => #_w1);
   IF #_w1 AND #Mod_TCP_Setup.Mod_Client[5].error THEN
       #Mod_TCP_Setup.Mod_Client[5].statusSave := #Mod_TCP_Setup.Mod_Client[5].status;
   END_IF;
END_REGION

REGION Network 16: Read Master-5 Coil Data Value
   RUNG wire#powerrail
      Contact( "AlwaysTRUE" )
      wire#w1
      Contact( #Mod_TCP_Setup.Mod_Client[5].request )
      Contact( #Mod_TCP_Setup.Mod_Client[5].busy )
      Move(in := 1, out1 => #PStep_No.MASTER_STEP_NO.Master_Step_No[5])
   END_RUNG
   RUNG wire#w1
      { S7_Templates := "SrcType := USInt" } EQ_Contact(in1 := #PStep_No.MASTER_STEP_NO.Master_Step_No[5], in2 := 1)
      Contact( #Mod_TCP_Setup.Mod_Client[5].done )
      wire#w2
      Move(in := "MODBUS_DATA_READ".MOD_RD_DEV_STN4[2].MOD_COIL_DATA, out1 => "MASTER_TCP_DATA".MOD_DEVICE_STATION4[2].MASTER_READ_DATA.MOD_COIL_DATA)
      R_Coil( #Mod_TCP_Setup.Mod_Client[5].request )
   END_RUNG
   RUNG wire#w2
      Move(in := 0, out1 => #PStep_No.MASTER_STEP_NO.Master_Step_No[5])
   END_RUNG
   RUNG wire#w2
      { S7_Templates := "SrcType := Int" } EQ_Contact(in1 := #LPG_Fill_Data.FILL_SEQ_OUT.Step_No, in2 := 3)
      { S7_Templates := "SrcType := USInt" } EQ_Contact(in1 := #PStep_No.MASTER_STEP_NO.Master_Step_No[6], in2 := 2)
      Move(in := 0, out1 => #PStep_No.MASTER_STEP_NO.Master_Step_No[6])
   END_RUNG
   // the same network as SCL:
   IF "AlwaysTRUE" AND #Mod_TCP_Setup.Mod_Client[5].request AND #Mod_TCP_Setup.Mod_Client[5].busy THEN
       #PStep_No.MASTER_STEP_NO.Master_Step_No[5] := 1;
   END_IF;
   #_w1 := "AlwaysTRUE" AND (#PStep_No.MASTER_STEP_NO.Master_Step_No[5] = 1) AND #Mod_TCP_Setup.Mod_Client[5].done;
   IF #_w1 THEN
       "MASTER_TCP_DATA".MOD_DEVICE_STATION4[2].MASTER_READ_DATA.MOD_COIL_DATA := "MODBUS_DATA_READ".MOD_RD_DEV_STN4[2].MOD_COIL_DATA;
       #Mod_TCP_Setup.Mod_Client[5].request := FALSE;
       #PStep_No.MASTER_STEP_NO.Master_Step_No[5] := 0;
   END_IF;
   IF #_w1 AND (#LPG_Fill_Data.FILL_SEQ_OUT.Step_No = 3) AND (#PStep_No.MASTER_STEP_NO.Master_Step_No[6] = 2) THEN
       #PStep_No.MASTER_STEP_NO.Master_Step_No[6] := 0;
   END_IF;
END_REGION

REGION Network 17: Write Coil Data
   // if multiple bit write not working
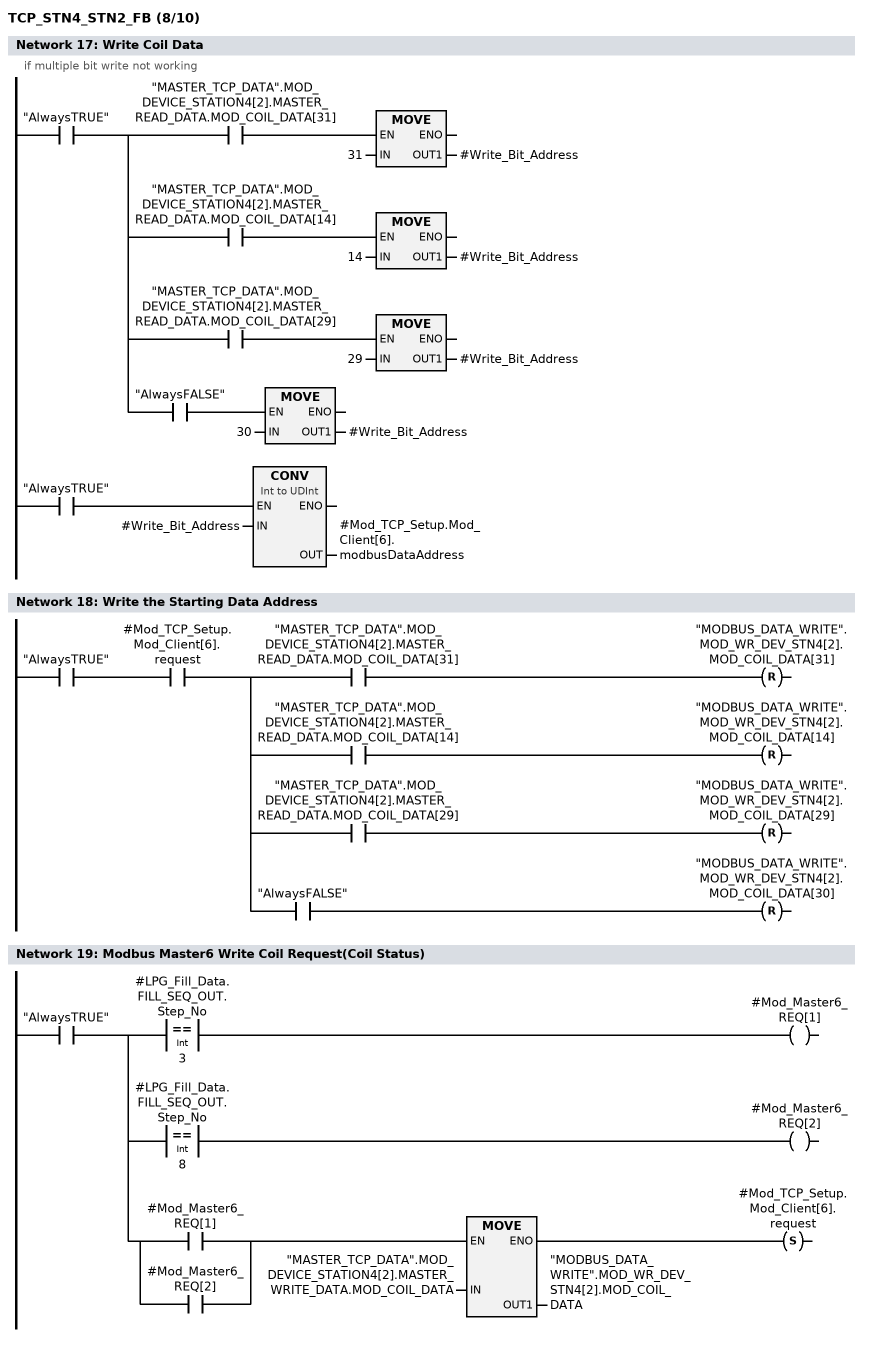
   RUNG wire#powerrail
      Contact( "AlwaysTRUE" )
      wire#w1
      Contact( "MASTER_TCP_DATA".MOD_DEVICE_STATION4[2].MASTER_READ_DATA.MOD_COIL_DATA[31] )
      Move(in := 31, out1 => #Write_Bit_Address)
   END_RUNG
   RUNG wire#w1
      Contact( "MASTER_TCP_DATA".MOD_DEVICE_STATION4[2].MASTER_READ_DATA.MOD_COIL_DATA[14] )
      Move(in := 14, out1 => #Write_Bit_Address)
   END_RUNG
   RUNG wire#w1
      Contact( "MASTER_TCP_DATA".MOD_DEVICE_STATION4[2].MASTER_READ_DATA.MOD_COIL_DATA[29] )
      Move(in := 29, out1 => #Write_Bit_Address)
   END_RUNG
   RUNG wire#w1
      Contact( "AlwaysFALSE" )
      Move(in := 30, out1 => #Write_Bit_Address)
   END_RUNG
   RUNG wire#powerrail
      Contact( "AlwaysTRUE" )
      { S7_Templates := "[SrcType := Int, DestType := UDInt]" } Convert(in := #Write_Bit_Address, out => #Mod_TCP_Setup.Mod_Client[6].modbusDataAddress)
   END_RUNG
   // the same network as SCL:
   IF "AlwaysTRUE" AND "MASTER_TCP_DATA".MOD_DEVICE_STATION4[2].MASTER_READ_DATA.MOD_COIL_DATA[31] THEN
       #Write_Bit_Address := 31;
   END_IF;
   IF "AlwaysTRUE" AND "MASTER_TCP_DATA".MOD_DEVICE_STATION4[2].MASTER_READ_DATA.MOD_COIL_DATA[14] THEN
       #Write_Bit_Address := 14;
   END_IF;
   IF "AlwaysTRUE" AND "MASTER_TCP_DATA".MOD_DEVICE_STATION4[2].MASTER_READ_DATA.MOD_COIL_DATA[29] THEN
       #Write_Bit_Address := 29;
   END_IF;
   IF "AlwaysTRUE" AND "AlwaysFALSE" THEN #Write_Bit_Address := 30; END_IF;
   IF "AlwaysTRUE" THEN
       #Mod_TCP_Setup.Mod_Client[6].modbusDataAddress := INT_TO_UDINT(#Write_Bit_Address);
   END_IF;
END_REGION

REGION Network 18: Write the Starting Data Address
   RUNG wire#powerrail
      Contact( "AlwaysTRUE" )
      Contact( #Mod_TCP_Setup.Mod_Client[6].request )
      wire#w1
      Contact( "MASTER_TCP_DATA".MOD_DEVICE_STATION4[2].MASTER_READ_DATA.MOD_COIL_DATA[31] )
      R_Coil( "MODBUS_DATA_WRITE".MOD_WR_DEV_STN4[2].MOD_COIL_DATA[31] )
   END_RUNG
   RUNG wire#w1
      Contact( "MASTER_TCP_DATA".MOD_DEVICE_STATION4[2].MASTER_READ_DATA.MOD_COIL_DATA[14] )
      R_Coil( "MODBUS_DATA_WRITE".MOD_WR_DEV_STN4[2].MOD_COIL_DATA[14] )
   END_RUNG
   RUNG wire#w1
      Contact( "MASTER_TCP_DATA".MOD_DEVICE_STATION4[2].MASTER_READ_DATA.MOD_COIL_DATA[29] )
      R_Coil( "MODBUS_DATA_WRITE".MOD_WR_DEV_STN4[2].MOD_COIL_DATA[29] )
   END_RUNG
   RUNG wire#w1
      Contact( "AlwaysFALSE" )
      R_Coil( "MODBUS_DATA_WRITE".MOD_WR_DEV_STN4[2].MOD_COIL_DATA[30] )
   END_RUNG
   // the same network as SCL:
   #_w1 := "AlwaysTRUE" AND #Mod_TCP_Setup.Mod_Client[6].request;
   IF #_w1 AND "MASTER_TCP_DATA".MOD_DEVICE_STATION4[2].MASTER_READ_DATA.MOD_COIL_DATA[31] THEN
       "MODBUS_DATA_WRITE".MOD_WR_DEV_STN4[2].MOD_COIL_DATA[31] := FALSE;
   END_IF;
   IF #_w1 AND "MASTER_TCP_DATA".MOD_DEVICE_STATION4[2].MASTER_READ_DATA.MOD_COIL_DATA[14] THEN
       "MODBUS_DATA_WRITE".MOD_WR_DEV_STN4[2].MOD_COIL_DATA[14] := FALSE;
   END_IF;
   IF #_w1 AND "MASTER_TCP_DATA".MOD_DEVICE_STATION4[2].MASTER_READ_DATA.MOD_COIL_DATA[29] THEN
       "MODBUS_DATA_WRITE".MOD_WR_DEV_STN4[2].MOD_COIL_DATA[29] := FALSE;
   END_IF;
   IF #_w1 AND "AlwaysFALSE" THEN "MODBUS_DATA_WRITE".MOD_WR_DEV_STN4[2].MOD_COIL_DATA[30] := FALSE; END_IF;
END_REGION

REGION Network 19: Modbus Master6 Write Coil Request(Coil Status)
   RUNG wire#powerrail
      Contact( "AlwaysTRUE" )
      wire#w1
      { S7_Templates := "SrcType := Int" } EQ_Contact(in1 := #LPG_Fill_Data.FILL_SEQ_OUT.Step_No, in2 := 3)
      Coil( #Mod_Master6_REQ[1] )
   END_RUNG
   RUNG wire#w1
      { S7_Templates := "SrcType := Int" } EQ_Contact(in1 := #LPG_Fill_Data.FILL_SEQ_OUT.Step_No, in2 := 8)
      Coil( #Mod_Master6_REQ[2] )
   END_RUNG
   RUNG wire#w1
      Contact( #Mod_Master6_REQ[1] )
      wire#w2
      Move(in := "MASTER_TCP_DATA".MOD_DEVICE_STATION4[2].MASTER_WRITE_DATA.MOD_COIL_DATA, out1 => "MODBUS_DATA_WRITE".MOD_WR_DEV_STN4[2].MOD_COIL_DATA)
      S_Coil( #Mod_TCP_Setup.Mod_Client[6].request )
   END_RUNG
   RUNG wire#w1
      Contact( #Mod_Master6_REQ[2] )
   END_RUNG wire#w2
   // the same network as SCL:
   #Mod_Master6_REQ[1] := "AlwaysTRUE" AND (#LPG_Fill_Data.FILL_SEQ_OUT.Step_No = 3);
   #Mod_Master6_REQ[2] := "AlwaysTRUE" AND (#LPG_Fill_Data.FILL_SEQ_OUT.Step_No = 8);
   IF "AlwaysTRUE" AND (#Mod_Master6_REQ[1] OR #Mod_Master6_REQ[2]) THEN
       "MODBUS_DATA_WRITE".MOD_WR_DEV_STN4[2].MOD_COIL_DATA := "MASTER_TCP_DATA".MOD_DEVICE_STATION4[2].MASTER_WRITE_DATA.MOD_COIL_DATA;
       #Mod_TCP_Setup.Mod_Client[6].request := TRUE;
   END_IF;
END_REGION

REGION Network 20: Modbus Master6 Write Coil Status
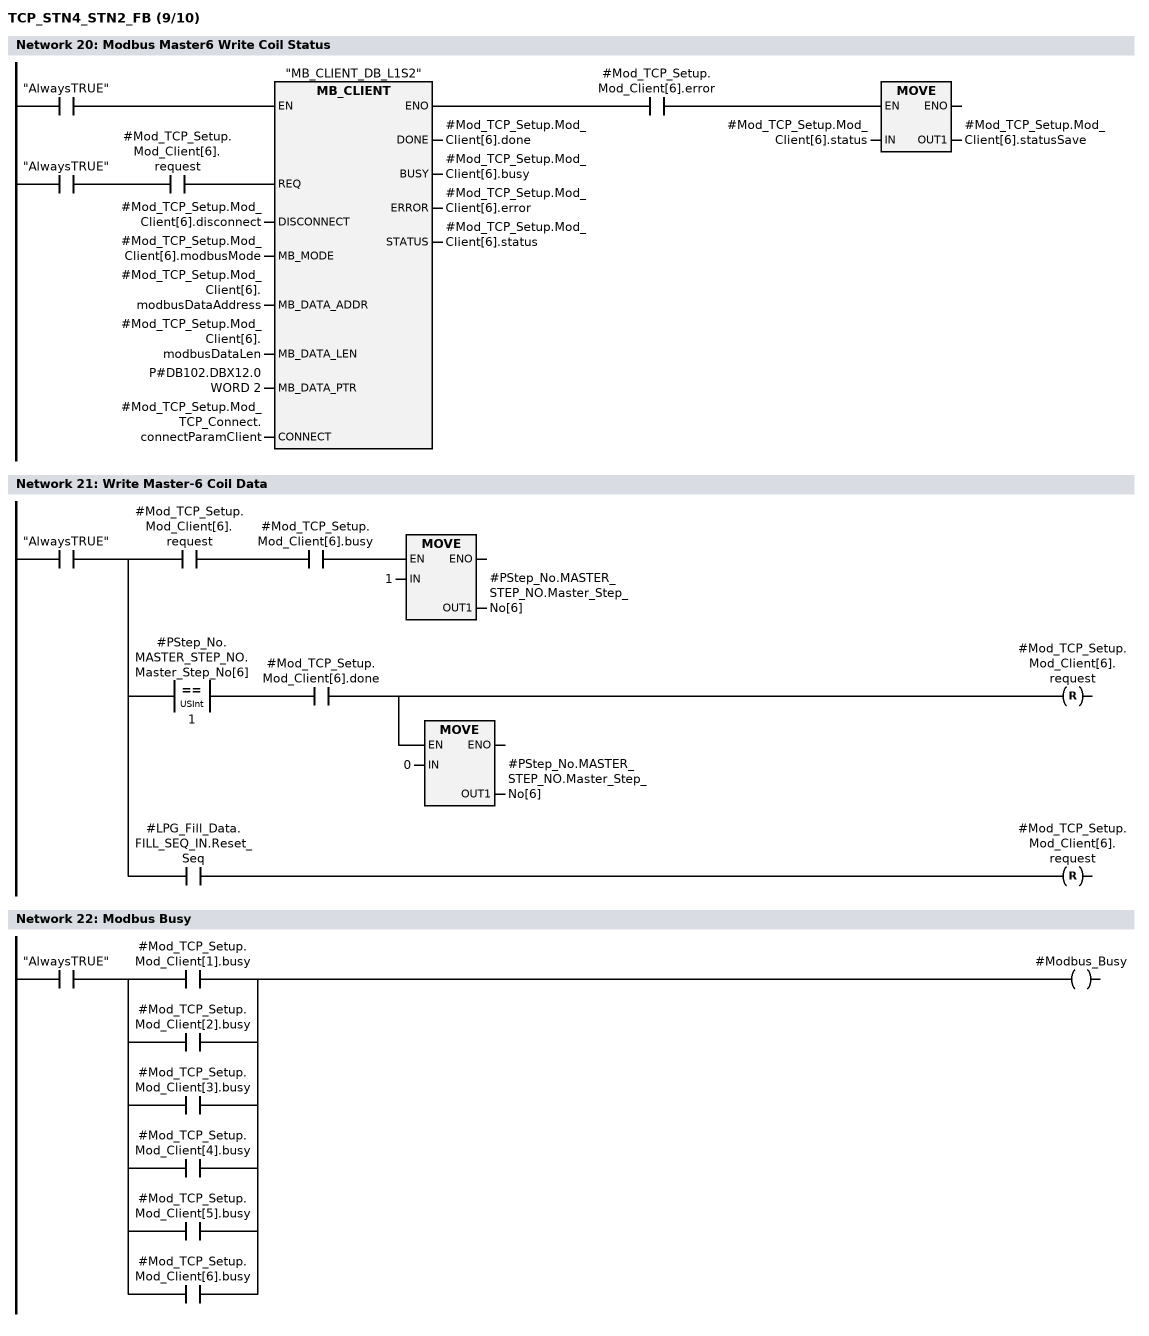
   RUNG wire#powerrail
      Contact( "AlwaysTRUE" )
      "MB_CLIENT_DB_L1S2".MB_CLIENT(REQ := wire#w1, DISCONNECT := #Mod_TCP_Setup.Mod_Client[6].disconnect, MB_MODE := #Mod_TCP_Setup.Mod_Client[6].modbusMode, MB_DATA_ADDR := #Mod_TCP_Setup.Mod_Client[6].modbusDataAddress, MB_DATA_LEN := #Mod_TCP_Setup.Mod_Client[6].modbusDataLen, MB_DATA_PTR := P#DB102.DBX12.0 WORD 2, CONNECT := #Mod_TCP_Setup.Mod_TCP_Connect.connectParamClient, DONE => #Mod_TCP_Setup.Mod_Client[6].done, BUSY => #Mod_TCP_Setup.Mod_Client[6].busy, ERROR => #Mod_TCP_Setup.Mod_Client[6].error, STATUS => #Mod_TCP_Setup.Mod_Client[6].status)
      Contact( #Mod_TCP_Setup.Mod_Client[6].error )
      Move(in := #Mod_TCP_Setup.Mod_Client[6].status, out1 => #Mod_TCP_Setup.Mod_Client[6].statusSave)
   END_RUNG
   RUNG wire#powerrail
      Contact( "AlwaysTRUE" )
      Contact( #Mod_TCP_Setup.Mod_Client[6].request )
   END_RUNG wire#w1
   // the same network as SCL:
   "MB_CLIENT_DB_L1S2"(EN := "AlwaysTRUE",   // MB_CLIENT
                       REQ := "AlwaysTRUE" AND #Mod_TCP_Setup.Mod_Client[6].request,
                       DISCONNECT := #Mod_TCP_Setup.Mod_Client[6].disconnect,
                       MB_MODE := #Mod_TCP_Setup.Mod_Client[6].modbusMode,
                       MB_DATA_ADDR := #Mod_TCP_Setup.Mod_Client[6].modbusDataAddress,
                       MB_DATA_LEN := #Mod_TCP_Setup.Mod_Client[6].modbusDataLen,
                       MB_DATA_PTR := P#DB102.DBX12.0 WORD 2,
                       CONNECT := #Mod_TCP_Setup.Mod_TCP_Connect.connectParamClient,
                       DONE => #Mod_TCP_Setup.Mod_Client[6].done,
                       BUSY => #Mod_TCP_Setup.Mod_Client[6].busy,
                       ERROR => #Mod_TCP_Setup.Mod_Client[6].error,
                       STATUS => #Mod_TCP_Setup.Mod_Client[6].status,
                       ENO => #_w1);
   IF #_w1 AND #Mod_TCP_Setup.Mod_Client[6].error THEN
       #Mod_TCP_Setup.Mod_Client[6].statusSave := #Mod_TCP_Setup.Mod_Client[6].status;
   END_IF;
END_REGION

REGION Network 21: Write Master-6 Coil Data
   RUNG wire#powerrail
      Contact( "AlwaysTRUE" )
      wire#w1
      Contact( #Mod_TCP_Setup.Mod_Client[6].request )
      Contact( #Mod_TCP_Setup.Mod_Client[6].busy )
      Move(in := 1, out1 => #PStep_No.MASTER_STEP_NO.Master_Step_No[6])
   END_RUNG
   RUNG wire#w1
      { S7_Templates := "SrcType := USInt" } EQ_Contact(in1 := #PStep_No.MASTER_STEP_NO.Master_Step_No[6], in2 := 1)
      Contact( #Mod_TCP_Setup.Mod_Client[6].done )
      wire#w2
      R_Coil( #Mod_TCP_Setup.Mod_Client[6].request )
   END_RUNG
   RUNG wire#w2
      Move(in := 0, out1 => #PStep_No.MASTER_STEP_NO.Master_Step_No[6])
   END_RUNG
   RUNG wire#w1
      Contact( #LPG_Fill_Data.FILL_SEQ_IN.Reset_Seq )
      R_Coil( #Mod_TCP_Setup.Mod_Client[6].request )
   END_RUNG
   // the same network as SCL:
   IF "AlwaysTRUE" AND #Mod_TCP_Setup.Mod_Client[6].request AND #Mod_TCP_Setup.Mod_Client[6].busy THEN
       #PStep_No.MASTER_STEP_NO.Master_Step_No[6] := 1;
   END_IF;
   #_w1 := "AlwaysTRUE" AND (#PStep_No.MASTER_STEP_NO.Master_Step_No[6] = 1) AND #Mod_TCP_Setup.Mod_Client[6].done;
   IF #_w1 THEN
       #Mod_TCP_Setup.Mod_Client[6].request := FALSE;
       #PStep_No.MASTER_STEP_NO.Master_Step_No[6] := 0;
   END_IF;
   IF "AlwaysTRUE" AND #LPG_Fill_Data.FILL_SEQ_IN.Reset_Seq THEN
       #Mod_TCP_Setup.Mod_Client[6].request := FALSE;
   END_IF;
END_REGION

REGION Network 22: Modbus Busy
   RUNG wire#powerrail
      Contact( "AlwaysTRUE" )
      wire#w1
      Contact( #Mod_TCP_Setup.Mod_Client[1].busy )
      wire#w2
      Coil( #Modbus_Busy )
   END_RUNG
   RUNG wire#w1
      Contact( #Mod_TCP_Setup.Mod_Client[2].busy )
   END_RUNG wire#w2
   RUNG wire#w1
      Contact( #Mod_TCP_Setup.Mod_Client[3].busy )
   END_RUNG wire#w2
   RUNG wire#w1
      Contact( #Mod_TCP_Setup.Mod_Client[4].busy )
   END_RUNG wire#w2
   RUNG wire#w1
      Contact( #Mod_TCP_Setup.Mod_Client[5].busy )
   END_RUNG wire#w2
   RUNG wire#w1
      Contact( #Mod_TCP_Setup.Mod_Client[6].busy )
   END_RUNG wire#w2
   // the same network as SCL:
   #Modbus_Busy := "AlwaysTRUE" AND (#Mod_TCP_Setup.Mod_Client[1].busy OR #Mod_TCP_Setup.Mod_Client[2].busy OR #Mod_TCP_Setup.Mod_Client[3].busy OR #Mod_TCP_Setup.Mod_Client[4].busy OR #Mod_TCP_Setup.Mod_Client[5].busy OR #Mod_TCP_Setup.Mod_Client[6].busy);
END_REGION

REGION Network 23
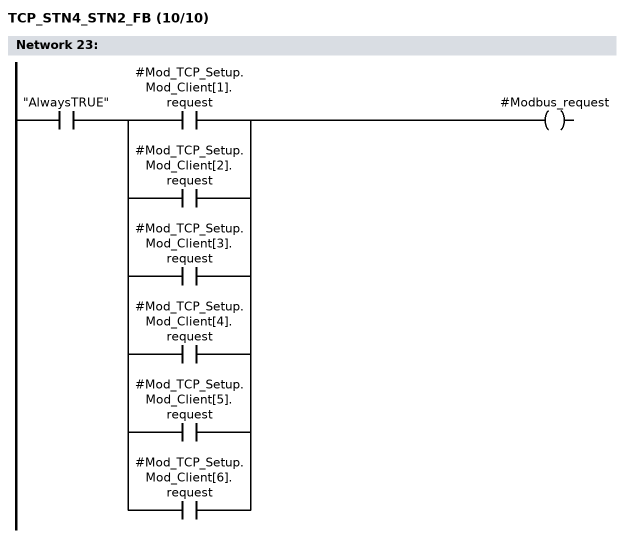
   RUNG wire#powerrail
      Contact( "AlwaysTRUE" )
      wire#w1
      Contact( #Mod_TCP_Setup.Mod_Client[1].request )
      wire#w2
      Coil( #Modbus_request )
   END_RUNG
   RUNG wire#w1
      Contact( #Mod_TCP_Setup.Mod_Client[2].request )
   END_RUNG wire#w2
   RUNG wire#w1
      Contact( #Mod_TCP_Setup.Mod_Client[3].request )
   END_RUNG wire#w2
   RUNG wire#w1
      Contact( #Mod_TCP_Setup.Mod_Client[4].request )
   END_RUNG wire#w2
   RUNG wire#w1
      Contact( #Mod_TCP_Setup.Mod_Client[5].request )
   END_RUNG wire#w2
   RUNG wire#w1
      Contact( #Mod_TCP_Setup.Mod_Client[6].request )
   END_RUNG wire#w2
   // the same network as SCL:
   #Modbus_request := "AlwaysTRUE" AND (#Mod_TCP_Setup.Mod_Client[1].request OR #Mod_TCP_Setup.Mod_Client[2].request OR #Mod_TCP_Setup.Mod_Client[3].request OR #Mod_TCP_Setup.Mod_Client[4].request OR #Mod_TCP_Setup.Mod_Client[5].request OR #Mod_TCP_Setup.Mod_Client[6].request);
END_REGION
END_FUNCTION_BLOCK
